{attribute 'qualified_only'}
VAR_GLOBAL	
	xOverride		:	BOOL := FALSE; // Global override of motion safety settings.
END_VAR

(* stored: Version 1.1.0.1, ProductVersion 3.1.4022.18
   GVL GVL: Id {981954b3-638a-42e3-8deb-b73c0db39eb1} *)
